// TIA Portal V19 export
TYPE "LAF_typeVfdGeneralParameters"
// stored: Access Published
   STRUCT
      refSpeed : Real := 1000.0;
      simActive : Bool;   // Manual mode parameters for axis control interface
      hwID : HW_IO;
      simulatePar : "LAF_typeVfdSimulateParameters";
   END_STRUCT;
END_TYPE
